TYPE OutputBase_10CEE7DE :
STRUCT
END_STRUCT
END_TYPE

(* stored: Version 1.2.0.0, ProductVersion 3.1.4024.11
   DUT OutputBase_10CEE7DE: Id {5ff4f419-1f40-4265-8028-f878d862bd7b} *)
